# EPICS substitutions: app/Db/gmb.substitutions
file gmb.template {
    { DEV = "$(DEV)" }
}
